Omron CX-Programmer project NewProject (CX-Programmer 9.73)

# PLC NewPLC1: CP1E N20

## Global symbols (name address type ; comment)
0.00 BOOL  ; senser
0.01 BOOL  ; reset
100.01 BOOL  ; motor
100.02 BOOL  ; lamp
100.03 BOOL  ; lamp 2
100.04 BOOL  ; lamp4
C001 BOOL  ; counter
T001 BOOL  ; timer
T002 BOOL  ; timer
T003 BOOL  ; timer

## Program NewProgram1 (cyclic task 0)

### Section Section1

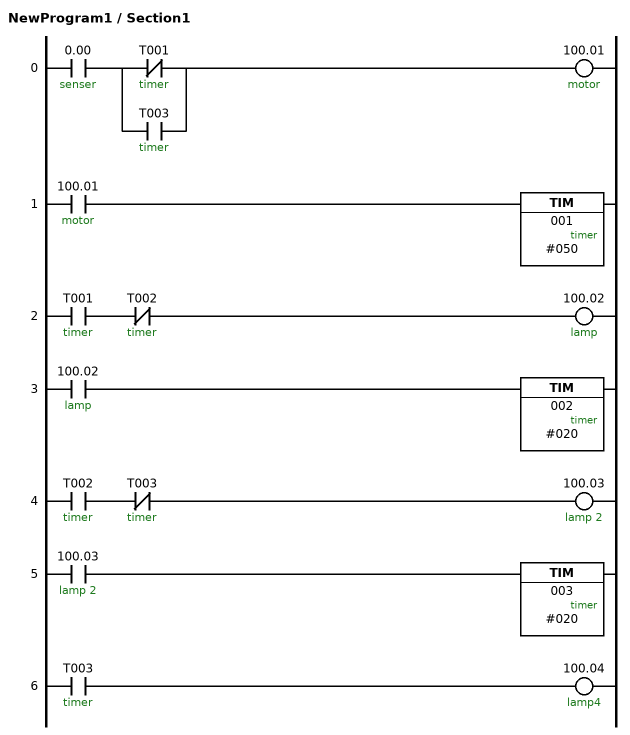
; rung 0
LD 0.00  ; senser
LDNOT T001  ; timer
OR T003  ; timer
ANDLD
OUT 100.01  ; motor
; rung 1
LD 100.01  ; motor
TIM 001 #050  ; timer
; rung 2
LD T001  ; timer
ANDNOT T002  ; timer
OUT 100.02  ; lamp
; rung 3
LD 100.02  ; lamp
TIM 002 #020  ; timer
; rung 4
LD T002  ; timer
ANDNOT T003  ; timer
OUT 100.03  ; lamp 2
; rung 5
LD 100.03  ; lamp 2
TIM 003 #020  ; timer
; rung 6
LD T003  ; timer
OUT 100.04  ; lamp4

### Section END
; rung 0
END(001)